KUKA KRL program: D15_DROPOFF05.src, D15_DROPOFF05.dat

--- D15_DROPOFF05.src ---
&ACCESS RVO
&REL 53
&COMMENT Drop To WeldStation4
&PARAM DISKPATH = KRC:\R1\Program\SbtComm001Main\D
DEF  D15_DROPOFF05 ( )
;********************************

;CREATOR : SPEEDBOT
;DATE    : 2024-09-23
;PROGRAM : sbtComm001_DDROPOFF05

;********************************
;FOLD INI;%{PE}
  ;FOLD BASISTECH INI
    GLOBAL INTERRUPT DECL 3 WHEN $STOPMESS==TRUE DO IR_STOPM ( )
    INTERRUPT ON 3
    BAS (#INITMOV,0 )
  ;ENDFOLD (BASISTECH INI)
  ;FOLD USER INI
    ;Make your modifications here
    continue
    if $MOVE_BCO == FALSE Then
      ; BCO
      ptp cur_jpos_()
    endif
  ;ENDFOLD (USER INI)
;ENDFOLD (INI)

;place example code
;waiting for PLC clearance to proceed
;FOLD PLC.RequestToContinue ;%{PE}
req_to_continue_()
;ENDFOLD
;FOLD PLC.PathSegment IN Segment Nr: 76 ;%{PE}
path_segment_(76)
;ENDFOLD
;entering interference zone 1 with robot *.
;Enter Zone With R***
;FOLD PLC.EnterZone IN Zone Nr: ZONE [1] ;%{PE}
zone_ctrl_(#I_ENTER, 1)
;ENDFOLD
;teach the robot to the placement point
;FOLD SPTP P1 CONT Vel=100 % PDAT1 Tool[1] Base[0] ;%{PE}
;FOLD Parameters ;%{h}
;Params IlfProvider=kukaroboter.basistech.inlineforms.movement.spline; Kuka.IsGlobalPoint=False; Kuka.PointName=P1; Kuka.BlendingEnabled=True; Kuka.MoveDataPtpName=PDAT1; Kuka.VelocityPtp=100; Kuka.VelocityFieldEnabled=True; Kuka.ColDetectFieldEnabled=True; Kuka.CurrentCDSetIndex=0; Kuka.MovementParameterFieldEnabled=True; IlfCommand=SPTP
;ENDFOLD
SPTP XP1 WITH $VEL_AXIS[1] = SVEL_JOINT(100.0), $TOOL = STOOL2(FP1), $BASE = SBASE(FP1.BASE_NO), $IPO_MODE = SIPO_MODE(FP1.IPO_FRAME), $LOAD = SLOAD(FP1.TOOL_NO), $ACC_AXIS[1] = SACC_JOINT(PPDAT1), $APO = SAPO_PTP(PPDAT1), $GEAR_JERK[1] = SGEAR_JERK(PPDAT1), $COLLMON_TOL_PRO[1] = USE_CM_PRO_VALUES(0) C_Spl
;ENDFOLD
;FOLD SPTP P2 CONT Vel=100 % PDAT2 Tool[1] Base[0] ;%{PE}
;FOLD Parameters ;%{h}
;Params IlfProvider=kukaroboter.basistech.inlineforms.movement.spline; Kuka.IsGlobalPoint=False; Kuka.PointName=P2; Kuka.BlendingEnabled=True; Kuka.MoveDataPtpName=PDAT2; Kuka.VelocityPtp=100; Kuka.VelocityFieldEnabled=True; Kuka.ColDetectFieldEnabled=True; Kuka.CurrentCDSetIndex=0; Kuka.MovementParameterFieldEnabled=True; IlfCommand=SPTP
;ENDFOLD
SPTP XP2 WITH $VEL_AXIS[1] = SVEL_JOINT(100.0), $TOOL = STOOL2(FP2), $BASE = SBASE(FP2.BASE_NO), $IPO_MODE = SIPO_MODE(FP2.IPO_FRAME), $LOAD = SLOAD(FP2.TOOL_NO), $ACC_AXIS[1] = SACC_JOINT(PPDAT2), $APO = SAPO_PTP(PPDAT2), $GEAR_JERK[1] = SGEAR_JERK(PPDAT2), $COLLMON_TOL_PRO[1] = USE_CM_PRO_VALUES(0) C_Spl
;ENDFOLD
;FOLD SLIN P_DropUp CONT Vel=0.8 m/s CPDAT1 Tool[1] Base[0] ;%{PE}
;FOLD Parameters ;%{h}
;Params IlfProvider=kukaroboter.basistech.inlineforms.movement.spline; Kuka.IsGlobalPoint=False; Kuka.PointName=P_DropUp; Kuka.BlendingEnabled=True; Kuka.MoveDataName=CPDAT1; Kuka.VelocityPath=0.8; Kuka.VelocityFieldEnabled=True; Kuka.ColDetectFieldEnabled=True; Kuka.CurrentCDSetIndex=0; Kuka.MovementParameterFieldEnabled=True; IlfCommand=SLIN
;ENDFOLD
SLIN XP_DropUp WITH $VEL = SVEL_CP(0.8, , LCPDAT1), $TOOL = STOOL2(FP_DropUp), $BASE = SBASE(FP_DropUp.BASE_NO), $IPO_MODE = SIPO_MODE(FP_DropUp.IPO_FRAME), $LOAD = SLOAD(FP_DropUp.TOOL_NO), $ACC = SACC_CP(LCPDAT1), $ORI_TYPE = SORI_TYP(LCPDAT1), $APO = SAPO(LCPDAT1), $JERK = SJERK(LCPDAT1), $COLLMON_TOL_PRO[1] = USE_CM_PRO_VALUES(0) C_Spl
;ENDFOLD
;reach the placement point
;FOLD SLIN P_Drop Vel=0.3 m/s CPDAT2 Tool[1] Base[0] ;%{PE}
;FOLD Parameters ;%{h}
;Params IlfProvider=kukaroboter.basistech.inlineforms.movement.spline; Kuka.IsGlobalPoint=False; Kuka.PointName=P_Drop; Kuka.BlendingEnabled=False; Kuka.MoveDataName=CPDAT2; Kuka.VelocityPath=0.3; Kuka.VelocityFieldEnabled=True; Kuka.ColDetectFieldEnabled=True; Kuka.CurrentCDSetIndex=0; Kuka.MovementParameterFieldEnabled=True; IlfCommand=SLIN
;ENDFOLD
SLIN XP_Drop WITH $VEL = SVEL_CP(0.3, , LCPDAT2), $TOOL = STOOL2(FP_Drop), $BASE = SBASE(FP_Drop.BASE_NO), $IPO_MODE = SIPO_MODE(FP_Drop.IPO_FRAME), $LOAD = SLOAD(FP_Drop.TOOL_NO), $ACC = SACC_CP(LCPDAT2), $ORI_TYPE = SORI_TYP(LCPDAT2), $APO = SAPO(LCPDAT2), $JERK = SJERK(LCPDAT2), $COLLMON_TOL_PRO[1] = USE_CM_PRO_VALUES(0)
;ENDFOLD

;Call the end-effector control program
;CALL End_Program()

;waiting for PLC clearance to proceed
;FOLD PLC.RequestToContinue ;%{PE}
req_to_continue_()
;ENDFOLD
;FOLD PLC.PathSegment IN Segment Nr: 77 ;%{PE}
path_segment_(77)
;ENDFOLD

;Teach to lift a certain distance
;FOLD SLIN P_DropUp CONT Vel=0.5 m/s CPDAT3 Tool[1] Base[0] ;%{PE}
;FOLD Parameters ;%{h}
;Params IlfProvider=kukaroboter.basistech.inlineforms.movement.spline; Kuka.IsGlobalPoint=False; Kuka.PointName=P_DropUp; Kuka.BlendingEnabled=True; Kuka.MoveDataName=CPDAT3; Kuka.VelocityPath=0.5; Kuka.VelocityFieldEnabled=True; Kuka.ColDetectFieldEnabled=True; Kuka.CurrentCDSetIndex=0; Kuka.MovementParameterFieldEnabled=True; IlfCommand=SLIN
;ENDFOLD
SLIN XP_DropUp WITH $VEL = SVEL_CP(0.5, , LCPDAT3), $TOOL = STOOL2(FP_DropUp), $BASE = SBASE(FP_DropUp.BASE_NO), $IPO_MODE = SIPO_MODE(FP_DropUp.IPO_FRAME), $LOAD = SLOAD(FP_DropUp.TOOL_NO), $ACC = SACC_CP(LCPDAT3), $ORI_TYPE = SORI_TYP(LCPDAT3), $APO = SAPO(LCPDAT3), $JERK = SJERK(LCPDAT3), $COLLMON_TOL_PRO[1] = USE_CM_PRO_VALUES(0) C_Spl
;ENDFOLD
;Sensor detection can be invoked here
;Confirm that it has been placed down
;CALL DetectionProcedure()

;waiting for PLC clearance to proceed
;FOLD PLC.RequestToContinue ;%{PE}
req_to_continue_()
;ENDFOLD
;FOLD PLC.PathSegment IN Segment Nr: 78 ;%{PE}
path_segment_(78)
;ENDFOLD

;Teach the placement and leave trajectory
;FOLD SLIN P7 CONT Vel=2 m/s CPDAT5 Tool[1] Base[0] ;%{PE}
;FOLD Parameters ;%{h}
;Params IlfProvider=kukaroboter.basistech.inlineforms.movement.spline; Kuka.IsGlobalPoint=False; Kuka.PointName=P7; Kuka.BlendingEnabled=True; Kuka.MoveDataName=CPDAT5; Kuka.VelocityPath=2; Kuka.VelocityFieldEnabled=True; Kuka.ColDetectFieldEnabled=True; Kuka.CurrentCDSetIndex=0; Kuka.MovementParameterFieldEnabled=True; IlfCommand=SLIN
;ENDFOLD
SLIN XP7 WITH $VEL = SVEL_CP(2.0, , LCPDAT5), $TOOL = STOOL2(FP7), $BASE = SBASE(FP7.BASE_NO), $IPO_MODE = SIPO_MODE(FP7.IPO_FRAME), $LOAD = SLOAD(FP7.TOOL_NO), $ACC = SACC_CP(LCPDAT5), $ORI_TYPE = SORI_TYP(LCPDAT5), $APO = SAPO(LCPDAT5), $JERK = SJERK(LCPDAT5), $COLLMON_TOL_PRO[1] = USE_CM_PRO_VALUES(0) C_Spl
;ENDFOLD

;FOLD SLIN P8 CONT Vel=2 m/s CPDAT6 Tool[1] Base[0] ;%{PE}
;FOLD Parameters ;%{h}
;Params IlfProvider=kukaroboter.basistech.inlineforms.movement.spline; Kuka.IsGlobalPoint=False; Kuka.PointName=P8; Kuka.BlendingEnabled=True; Kuka.MoveDataName=CPDAT6; Kuka.VelocityPath=2; Kuka.VelocityFieldEnabled=True; Kuka.ColDetectFieldEnabled=True; Kuka.CurrentCDSetIndex=0; Kuka.MovementParameterFieldEnabled=True; IlfCommand=SLIN
;ENDFOLD
SLIN XP8 WITH $VEL = SVEL_CP(2.0, , LCPDAT6), $TOOL = STOOL2(FP8), $BASE = SBASE(FP8.BASE_NO), $IPO_MODE = SIPO_MODE(FP8.IPO_FRAME), $LOAD = SLOAD(FP8.TOOL_NO), $ACC = SACC_CP(LCPDAT6), $ORI_TYPE = SORI_TYP(LCPDAT6), $APO = SAPO(LCPDAT6), $JERK = SJERK(LCPDAT6), $COLLMON_TOL_PRO[1] = USE_CM_PRO_VALUES(0) C_Spl
;ENDFOLD
;FOLD SPTP P9 CONT Vel=100 % PDAT3 Tool[1] Base[0] ;%{PE}
;FOLD Parameters ;%{h}
;Params IlfProvider=kukaroboter.basistech.inlineforms.movement.spline; Kuka.IsGlobalPoint=False; Kuka.PointName=P9; Kuka.BlendingEnabled=True; Kuka.MoveDataPtpName=PDAT3; Kuka.VelocityPtp=100; Kuka.VelocityFieldEnabled=True; Kuka.ColDetectFieldEnabled=True; Kuka.CurrentCDSetIndex=0; Kuka.MovementParameterFieldEnabled=True; IlfCommand=SPTP
;ENDFOLD
SPTP XP9 WITH $VEL_AXIS[1] = SVEL_JOINT(100.0), $TOOL = STOOL2(FP9), $BASE = SBASE(FP9.BASE_NO), $IPO_MODE = SIPO_MODE(FP9.IPO_FRAME), $LOAD = SLOAD(FP9.TOOL_NO), $ACC_AXIS[1] = SACC_JOINT(PPDAT3), $APO = SAPO_PTP(PPDAT3), $GEAR_JERK[1] = SGEAR_JERK(PPDAT3), $COLLMON_TOL_PRO[1] = USE_CM_PRO_VALUES(0) C_Spl
;ENDFOLD
;FOLD SPTP P10 CONT Vel=100 % PDAT4 Tool[1] Base[0] ;%{PE}
;FOLD Parameters ;%{h}
;Params IlfProvider=kukaroboter.basistech.inlineforms.movement.spline; Kuka.IsGlobalPoint=False; Kuka.PointName=P10; Kuka.BlendingEnabled=True; Kuka.MoveDataPtpName=PDAT4; Kuka.VelocityPtp=100; Kuka.VelocityFieldEnabled=True; Kuka.ColDetectFieldEnabled=True; Kuka.CurrentCDSetIndex=0; Kuka.MovementParameterFieldEnabled=True; IlfCommand=SPTP
;ENDFOLD
SPTP XP10 WITH $VEL_AXIS[1] = SVEL_JOINT(100.0), $TOOL = STOOL2(FP10), $BASE = SBASE(FP10.BASE_NO), $IPO_MODE = SIPO_MODE(FP10.IPO_FRAME), $LOAD = SLOAD(FP10.TOOL_NO), $ACC_AXIS[1] = SACC_JOINT(PPDAT4), $APO = SAPO_PTP(PPDAT4), $GEAR_JERK[1] = SGEAR_JERK(PPDAT4), $COLLMON_TOL_PRO[1] = USE_CM_PRO_VALUES(0) C_Spl
;ENDFOLD
;This position has been fully cleared
;Does not interfere with the gripper and the corresponding robot.

;Report placement complete
;FOLD PLC.PathSegment IN Segment Nr: 79 ;%{PE}
path_segment_(79)
;ENDFOLD

;Exit the interference zone 1 with robot *.
;Enter Zone With R***
;FOLD PLC.ExitZone IN Zone Nr: ZONE [1] ;%{PE}
zone_ctrl_(#I_EXIT, 1)
;ENDFOLD


END

--- D15_DROPOFF05.dat ---
&ACCESS RVO
&REL 53
&COMMENT Drop To WeldStation4
&PARAM DISKPATH = KRC:\R1\Program\SbtComm001Main\D
DEFDAT  D15_DROPOFF05
;FOLD EXTERNAL DECLARATIONS;%{PE}%MKUKATPBASIS,%CEXT,%VCOMMON,%P
;FOLD BASISTECH EXT;%{PE}%MKUKATPBASIS,%CEXT,%VEXT,%P
EXT  BAS (BAS_COMMAND  :IN,REAL  :IN )
;ENDFOLD (BASISTECH EXT)
;FOLD USER EXT;%{E}%MKUKATPUSER,%CEXT,%VEXT,%P
;Make your modifications here

;ENDFOLD (USER EXT)
;ENDFOLD (EXTERNAL DECLARATIONS)
DECL MODULEPARAM_T LAST_TP_PARAMS={PARAMS[] "PLC.SEGMENTID=79; PLC.ZONEID=1; Kuka.VelocityFieldEnabled=True; Kuka.ColDetectFieldEnabled=True; Kuka.MovementParameterFieldEnabled=True; Kuka.IsAngleEnabled=False; Kuka.PointName=P_DropUp; Kuka.FrameData.base_no=0; Kuka.FrameData.tool_no=1; Kuka.FrameData.ipo_frame=#BASE; Kuka.isglobalpoint=False; Kuka.MoveDataPtpName=PDAT4; Kuka.MovementDataPdat.apo_mode=#CDIS; Kuka.MovementDataPdat.apo_dist=500; Kuka.MovementData.vel=0.5; Kuka.MovementData.acc=100; Kuka.MovementData.gear_jerk=100; Kuka.MovementData.exax_ign=0; Kuka.VelocityPtp=100; Kuka.BlendingEnabled=True; Kuka.CurrentCDSetIndex=0; Kuka.MoveDataName=CPDAT3; Kuka.MovementData.apo_fac=50; Kuka.MovementData.apo_dist=500; Kuka.MovementData.axis_acc=100; Kuka.MovementData.axis_vel=100; Kuka.MovementData.circ_typ=#BASE; Kuka.MovementData.jerk_fac=50; Kuka.MovementData.ori_typ=#VAR; Kuka.VelocityPath=0.5; Kuka.FrameData.point2=; BASIC.FRAMENAME=Frame1; BASIC.X_=0; BASIC.Y_=0; BASIC.Z_=-200; BASIC.A_=0; BASIC.B_=0; BASIC.C_=0; BASIC.SOURCENAME=P_Drop; BASIC.OFFSFRAME=Frame1; BASIC.OFFSETNAME=P_DropUp; SBTCOMM001.SLEEPTIME=1; SBTCOMM001.EVENTINTPRM1=5; SBTCOMM001.EVENTINTPRM2=1; SBTCOMM001.EVENTFLOATPRM1=4; SBTCOMM001.EVENTFLOATPRM2=0; SBTCOMM001.EVENTFLOATPRM3=0; SBTCOMM001.EVENTFLOATPRM4=0; SBTCOMM001.EVENTFLOATPRM5=0; SBTCOMM001.EVENTFLOATPRM6=0"}
DECL E6POS XP1={X 0.0,Y 0.0,Z 0.0,A 0.0,B 0.0,C 0.0,S 0,T 0,E1 0.0,E2 0.0,E3 0.0,E4 0.0,E5 0.0,E6 0.0}
DECL FDAT FP1={TOOL_NO 1,BASE_NO 0,IPO_FRAME #BASE,POINT2[] " "}
DECL PDAT PPDAT1={VEL 100.000,ACC 100.000,APO_DIST 500.000,APO_MODE #CDIS,GEAR_JERK 100.000,EXAX_IGN 0}
DECL E6POS XP2={X 0.0,Y 0.0,Z 0.0,A 0.0,B 0.0,C 0.0,S 0,T 0,E1 0.0,E2 0.0,E3 0.0,E4 0.0,E5 0.0,E6 0.0}
DECL FDAT FP2={TOOL_NO 1,BASE_NO 0,IPO_FRAME #BASE,POINT2[] " "}
DECL PDAT PPDAT2={VEL 100.000,ACC 100.000,APO_DIST 500.000,APO_MODE #CDIS,GEAR_JERK 100.000,EXAX_IGN 0}
DECL E6POS XP3={X 0.0,Y 0.0,Z 0.0,A 0.0,B 0.0,C 0.0,S 0,T 0,E1 0.0,E2 0.0,E3 0.0,E4 0.0,E5 0.0,E6 0.0}
DECL FDAT FP3={TOOL_NO 1,BASE_NO 0,IPO_FRAME #BASE,POINT2[] " "}
DECL LDAT LCPDAT1={VEL 0.800000,ACC 100.000,APO_DIST 500.000,APO_FAC 50.0000,AXIS_VEL 100.000,AXIS_ACC 100.000,ORI_TYP #VAR,CIRC_TYP #BASE,JERK_FAC 50.0000,GEAR_JERK 100.000,EXAX_IGN 0}
DECL E6POS XP4={X 0.0,Y 0.0,Z 0.0,A 0.0,B 0.0,C 0.0,S 0,T 0,E1 0.0,E2 0.0,E3 0.0,E4 0.0,E5 0.0,E6 0.0}
DECL FDAT FP4={TOOL_NO 1,BASE_NO 0,IPO_FRAME #BASE,POINT2[] " "}
DECL LDAT LCPDAT2={VEL 0.300000,ACC 100.000,APO_DIST 500.000,APO_FAC 50.0000,AXIS_VEL 100.000,AXIS_ACC 100.000,ORI_TYP #VAR,CIRC_TYP #BASE,JERK_FAC 50.0000,GEAR_JERK 100.000,EXAX_IGN 0}
DECL E6POS XP5={X 0.0,Y 0.0,Z 0.0,A 0.0,B 0.0,C 0.0,S 0,T 0,E1 0.0,E2 0.0,E3 0.0,E4 0.0,E5 0.0,E6 0.0}
DECL FDAT FP5={TOOL_NO 1,BASE_NO 0,IPO_FRAME #BASE,POINT2[] " "}
DECL LDAT LCPDAT3={VEL 0.500000,ACC 100.000,APO_DIST 500.000,APO_FAC 50.0000,AXIS_VEL 100.000,AXIS_ACC 100.000,ORI_TYP #VAR,CIRC_TYP #BASE,JERK_FAC 50.0000,GEAR_JERK 100.000,EXAX_IGN 0}
DECL E6POS XP6={X 0.0,Y 0.0,Z 0.0,A 0.0,B 0.0,C 0.0,S 0,T 0,E1 0.0,E2 0.0,E3 0.0,E4 0.0,E5 0.0,E6 0.0}
DECL FDAT FP6={TOOL_NO 1,BASE_NO 0,IPO_FRAME #BASE,POINT2[] " "}
DECL LDAT LCPDAT4={VEL 2.00000,ACC 100.000,APO_DIST 500.000,APO_FAC 50.0000,AXIS_VEL 100.000,AXIS_ACC 100.000,ORI_TYP #VAR,CIRC_TYP #BASE,JERK_FAC 50.0000,GEAR_JERK 100.000,EXAX_IGN 0}
DECL E6POS XP7={X 0.0,Y 0.0,Z 0.0,A 0.0,B 0.0,C 0.0,S 0,T 0,E1 0.0,E2 0.0,E3 0.0,E4 0.0,E5 0.0,E6 0.0}
DECL FDAT FP7={TOOL_NO 1,BASE_NO 0,IPO_FRAME #BASE,POINT2[] " "}
DECL LDAT LCPDAT5={VEL 0.00100000,ACC 100.000,APO_DIST 500.000,APO_FAC 50.0000,AXIS_VEL 100.000,AXIS_ACC 100.000,ORI_TYP #VAR,CIRC_TYP #BASE,JERK_FAC 50.0000,GEAR_JERK 100.000,EXAX_IGN 0}
DECL E6POS XP8={X 0.0,Y 0.0,Z 0.0,A 0.0,B 0.0,C 0.0,S 0,T 0,E1 0.0,E2 0.0,E3 0.0,E4 0.0,E5 0.0,E6 0.0}
DECL FDAT FP8={TOOL_NO 1,BASE_NO 0,IPO_FRAME #BASE,POINT2[] " "}
DECL LDAT LCPDAT6={VEL 2.00000,ACC 100.000,APO_DIST 500.000,APO_FAC 50.0000,AXIS_VEL 100.000,AXIS_ACC 100.000,ORI_TYP #VAR,CIRC_TYP #BASE,JERK_FAC 50.0000,GEAR_JERK 100.000,EXAX_IGN 0}
DECL E6POS XP9={X 0.0,Y 0.0,Z 0.0,A 0.0,B 0.0,C 0.0,S 0,T 0,E1 0.0,E2 0.0,E3 0.0,E4 0.0,E5 0.0,E6 0.0}
DECL FDAT FP9={TOOL_NO 1,BASE_NO 0,IPO_FRAME #BASE,POINT2[] " "}
DECL PDAT PPDAT3={VEL 100.000,ACC 100.000,APO_DIST 500.000,APO_MODE #CDIS,GEAR_JERK 100.000,EXAX_IGN 0}
DECL E6POS XP10={X 0.0,Y 0.0,Z 0.0,A 0.0,B 0.0,C 0.0,S 0,T 0,E1 0.0,E2 0.0,E3 0.0,E4 0.0,E5 0.0,E6 0.0}
DECL FDAT FP10={TOOL_NO 1,BASE_NO 0,IPO_FRAME #BASE,POINT2[] " "}
DECL PDAT PPDAT4={VEL 100.000,ACC 100.000,APO_DIST 500.000,APO_MODE #CDIS,GEAR_JERK 100.000,EXAX_IGN 0}
DECL E6POS XTeachP_Drop={X 0.0,Y 0.0,Z 0.0,A 0.0,B 0.0,C 0.0,S 0,T 0,E1 0.0,E2 0.0,E3 0.0,E4 0.0,E5 0.0,E6 0.0}
DECL FDAT FTeachP_Drop={TOOL_NO 1,BASE_NO 0,IPO_FRAME #BASE,POINT2[] " "}
DECL E6POS XP_DropUp={X 0.0,Y 0.0,Z 0.0,A 0.0,B 0.0,C 0.0,S 0,T 0,E1 0.0,E2 0.0,E3 0.0,E4 0.0,E5 0.0,E6 0.0}
DECL FDAT FP_DropUp={TOOL_NO 1,BASE_NO 0,IPO_FRAME #BASE,POINT2[] " "}
DECL E6POS XP_Drop={X -653.378418,Y 1492.82825,Z 1786.65149,A -58.7324829,B 23.3739033,C -179.497070,S 2,T 11,E1 0.0,E2 0.0,E3 0.0,E4 0.0,E5 0.0,E6 0.0}
DECL FDAT FP_Drop={TOOL_NO 1,BASE_NO 0,IPO_FRAME #BASE,POINT2[] " "}
DECL FRAME Frame1={X 0.0,Y 0.0,Z 0.0,A 0.0,B 0.0,C 0.0}
ENDDAT
